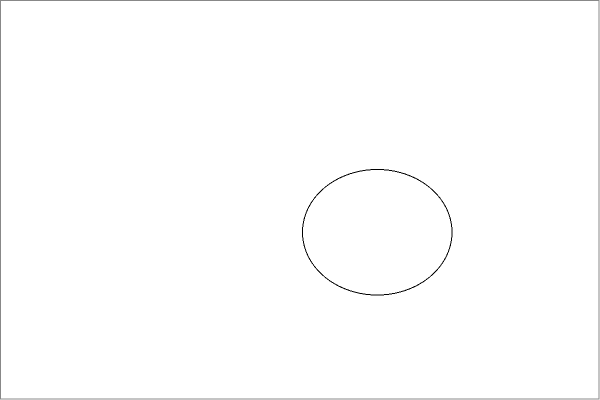
VISUALIZATION vPISTONS  // 600x400
    Ellipse (302,169 150x126)
END_VISUALIZATION

(* stored: Version 1.1.0.1, ProductVersion 3.1.4024.12
   Visu vPISTONS: Id {e8bda441-e226-4bf5-a4e7-de24e81be300} *)
